(* PLC project x *)

PROGRAM FBD_B
  VAR
    ctr : CTU;
  END_VAR
  VAR  (* added by the conversion: wires and edge detectors of the diagram *)
    R_TRIG1 : R_TRIG;
    _AND52_OUT : BOOL;
  END_VAR

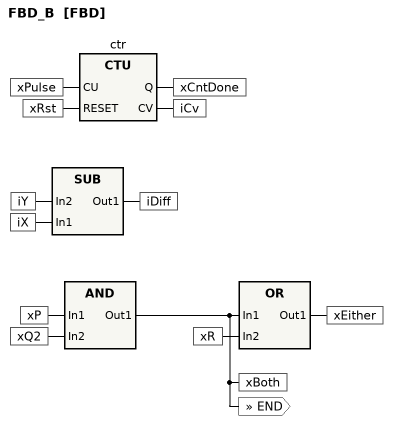
(* FBD diagram, written out as Structured Text *)
R_TRIG1(CLK := xPulse);
ctr(CU := R_TRIG1.Q, RESET := xRst, CV => iCv);
xCntDone := ctr.Q;
iDiff := iY - iX;
_AND52_OUT := xP AND xQ2;
xBoth := _AND52_OUT;
xEither := _AND52_OUT OR xR;
IF _AND52_OUT THEN JMP END; END_IF;
END_PROGRAM
